// TIA Portal V18 export
// export: Created 2025-12-01T17:53:15.9453864Z, ExportSetting None, DisplayName Totally Integrated Automation Portal, DisplayVersion V18 Update 5, DisplayName TIA Portal Openness, DisplayVersion V18 Update 5, DisplayName TIA Portal Teamcenter Gateway, DisplayVersion V18, DisplayName TIA Portal Version Control Interface, DisplayVersion V18, DisplayName STEP 7 Professional, DisplayVersion V18 Update 5, DisplayName STEP 7 Safety, DisplayVersion V18, DisplayName WinCC Professional, DisplayVersion V18 Update 5
Screen "440PartData1"  1280x800, Number=440, Template=04Information
  ScreenLayer 
    FaceplateInstance "PartData_HMI_1" at 0,87 size 1280x600  FaceplateTypeName=500 User@$@104 PartDataManage@$@104.2 HMI@$@PartData_HMI V 0.0.14
